TYPE ST_MagnetLiftSys :
STRUCT
END_STRUCT
END_TYPE

(* stored: Version 1.1.0.1, ProductVersion 3.1.4024.12
   DUT ST_MagnetLiftSys: Id {ad5393ca-1dea-4eaf-88c9-f406d31feb5c} *)
